TYPE INTERNAL PushoverRequest :
STRUCT
  TokenLength : INT;
  UserLength : INT;
  TitleLength : INT;  
  MessageLength : INT;
  DeviceLength : INT;
  UrlLength : INT;
  UrlTitleLength : INT;
  CallbackLength : INT;  
  ProxyHostLength : INT;  
  
  Retry : INT;
  Expire : INT;  
  MessageType : PushoverMessageType;  
  Priority : PushoverPriority;
  Sound : PushoverSound;
  Timestamp : INT; //< UNIX Timestamp in seconds 
  TimeToLive : INT; //< in seconds
  ProxyPort : INT;

  Token : STRING(80);
  User : STRING(80);  
  Device : STRING(80);
  Url : STRING(511);  
  UrlTitle : STRING(99);
  Callback : STRING(255);
  ProxyHost : STRING(80);
  Title : STRING(249);  
  Message : STRING(1023);  
END_STRUCT
END_TYPE

(* stored: Version 1.1.0.1, ProductVersion 3.1.4024.12
   DUT PushoverRequest: Id {f17a5064-8416-4c04-9856-ade6756db10d} *)
